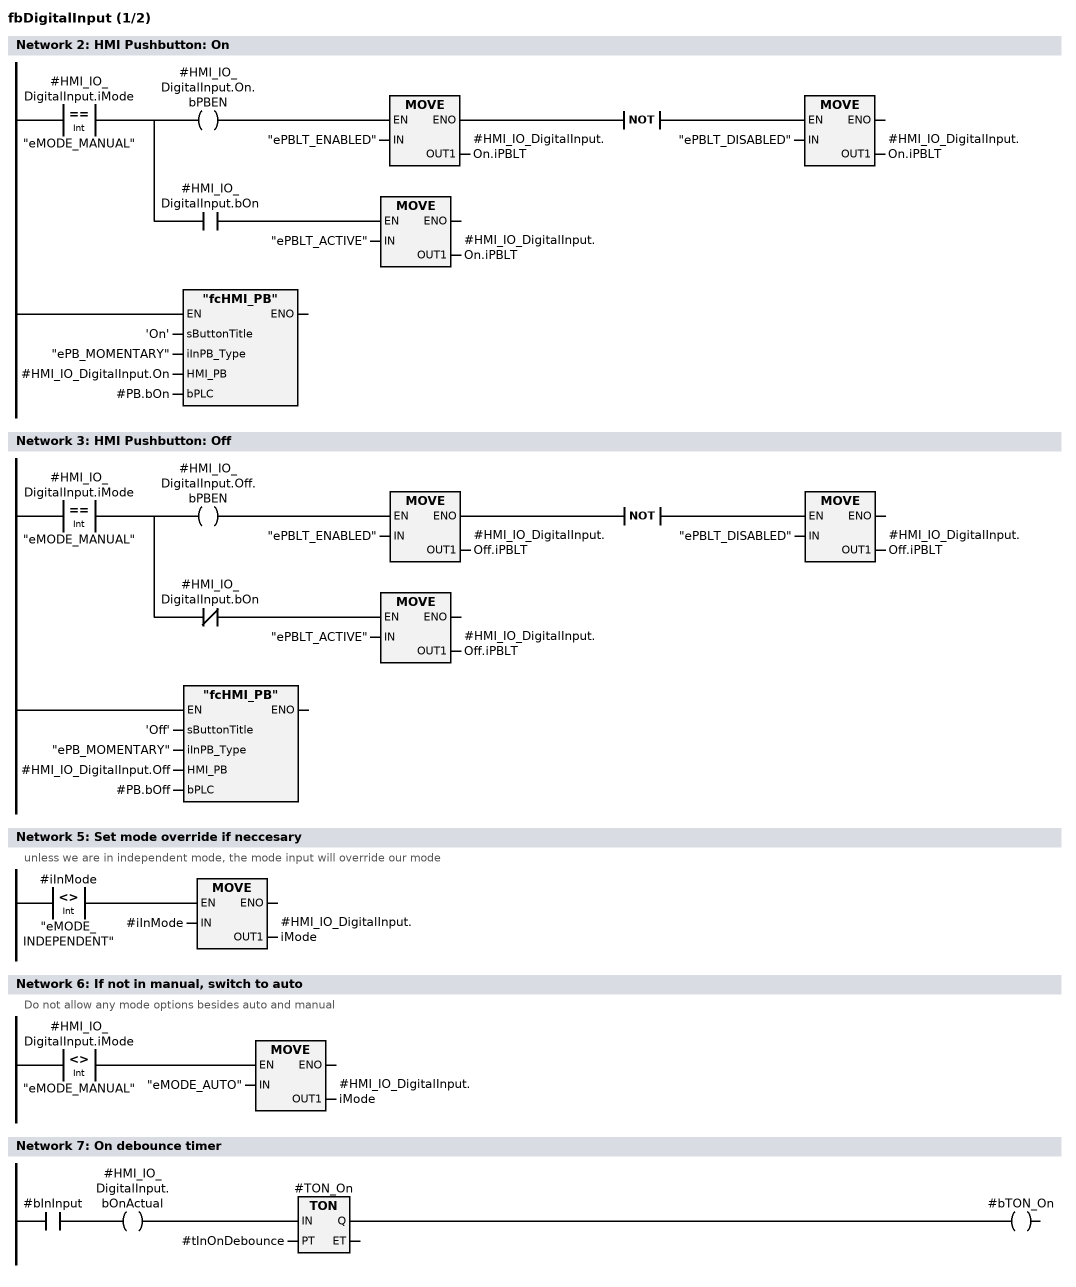
   RUNG wire#powerrail
      { S7_Templates := "SrcType := Int" } EQ_Contact(in1 := #HMI_IO_DigitalInput.iMode, in2 := "eMODE_MANUAL")
      wire#w1
      Coil( #HMI_IO_DigitalInput.On.bPBEN )
      Move(in := "ePBLT_ENABLED", out1 => #HMI_IO_DigitalInput.On.iPBLT)
      Not()
      Move(in := "ePBLT_DISABLED", out1 => #HMI_IO_DigitalInput.On.iPBLT)
   END_RUNG
   RUNG wire#w1
      Contact( #HMI_IO_DigitalInput.bOn )
      Move(in := "ePBLT_ACTIVE", out1 => #HMI_IO_DigitalInput.On.iPBLT)
   END_RUNG
   RUNG wire#powerrail
      "fcHMI_PB"(sButtonTitle := 'On', iInPB_Type := "ePB_MOMENTARY", HMI_PB := #HMI_IO_DigitalInput.On, bPLC := #PB.bOn)
   END_RUNG
   // the same network as SCL:
   #HMI_IO_DigitalInput.On.bPBEN := #HMI_IO_DigitalInput.iMode = "eMODE_MANUAL";
   IF #HMI_IO_DigitalInput.On.bPBEN THEN #HMI_IO_DigitalInput.On.iPBLT := "ePBLT_ENABLED"; END_IF;
   IF NOT #HMI_IO_DigitalInput.On.bPBEN THEN #HMI_IO_DigitalInput.On.iPBLT := "ePBLT_DISABLED"; END_IF;
   IF #HMI_IO_DigitalInput.On.bPBEN AND #HMI_IO_DigitalInput.bOn THEN
       #HMI_IO_DigitalInput.On.iPBLT := "ePBLT_ACTIVE";
   END_IF;
   "fcHMI_PB"(sButtonTitle := 'On',
              iInPB_Type := "ePB_MOMENTARY",
              HMI_PB := #HMI_IO_DigitalInput.On,
              bPLC := #PB.bOn);
END_REGION

REGION Network 3: HMI Pushbutton: Off
   RUNG wire#powerrail
      { S7_Templates := "SrcType := Int" } EQ_Contact(in1 := #HMI_IO_DigitalInput.iMode, in2 := "eMODE_MANUAL")
      wire#w1
      Coil( #HMI_IO_DigitalInput.Off.bPBEN )
      Move(in := "ePBLT_ENABLED", out1 => #HMI_IO_DigitalInput.Off.iPBLT)
      Not()
      Move(in := "ePBLT_DISABLED", out1 => #HMI_IO_DigitalInput.Off.iPBLT)
   END_RUNG
   RUNG wire#w1
      I_Contact( #HMI_IO_DigitalInput.bOn )
      Move(in := "ePBLT_ACTIVE", out1 => #HMI_IO_DigitalInput.Off.iPBLT)
   END_RUNG
   RUNG wire#powerrail
      "fcHMI_PB"(sButtonTitle := 'Off', iInPB_Type := "ePB_MOMENTARY", HMI_PB := #HMI_IO_DigitalInput.Off, bPLC := #PB.bOff)
   END_RUNG
   // the same network as SCL:
   #HMI_IO_DigitalInput.Off.bPBEN := #HMI_IO_DigitalInput.iMode = "eMODE_MANUAL";
   IF #HMI_IO_DigitalInput.Off.bPBEN THEN #HMI_IO_DigitalInput.Off.iPBLT := "ePBLT_ENABLED"; END_IF;
   IF NOT #HMI_IO_DigitalInput.Off.bPBEN THEN #HMI_IO_DigitalInput.Off.iPBLT := "ePBLT_DISABLED"; END_IF;
   IF #HMI_IO_DigitalInput.Off.bPBEN AND NOT #HMI_IO_DigitalInput.bOn THEN
       #HMI_IO_DigitalInput.Off.iPBLT := "ePBLT_ACTIVE";
   END_IF;
   "fcHMI_PB"(sButtonTitle := 'Off',
              iInPB_Type := "ePB_MOMENTARY",
              HMI_PB := #HMI_IO_DigitalInput.Off,
              bPLC := #PB.bOff);
END_REGION

REGION Network 4: --------------------------------------------------- Control Logic ------------------------------------------------------------
END_REGION

REGION Network 5: Set mode override if neccesary
   // unless we are in independent mode, the mode input will override our mode
   RUNG wire#powerrail
      { S7_Templates := "SrcType := Int" } NE_Contact(in1 := #iInMode, in2 := "eMODE_INDEPENDENT")
      { S7_GenerateENO := "TRUE" } Move(in := #iInMode, out1 => #HMI_IO_DigitalInput.iMode)
   END_RUNG
   // the same network as SCL:
   IF #iInMode <> "eMODE_INDEPENDENT" THEN #HMI_IO_DigitalInput.iMode := #iInMode; END_IF;
END_REGION

REGION Network 6: If not in manual, switch to auto
   // Do not allow any mode options besides auto and manual
   RUNG wire#powerrail
      { S7_Templates := "SrcType := Int" } NE_Contact(in1 := #HMI_IO_DigitalInput.iMode, in2 := "eMODE_MANUAL")
      Move(in := "eMODE_AUTO", out1 => #HMI_IO_DigitalInput.iMode)
   END_RUNG
   // the same network as SCL:
   IF #HMI_IO_DigitalInput.iMode <> "eMODE_MANUAL" THEN #HMI_IO_DigitalInput.iMode := "eMODE_AUTO"; END_IF;
END_REGION

REGION Network 7: On debounce timer
   #HMI_IO_DigitalInput.bOnActual := #bInInput;
   #TON_On.TON(IN := #bInInput, PT := #tInOnDebounce);
   #bTON_On := #TON_On.Q;
END_REGION

REGION Network 8: On logic
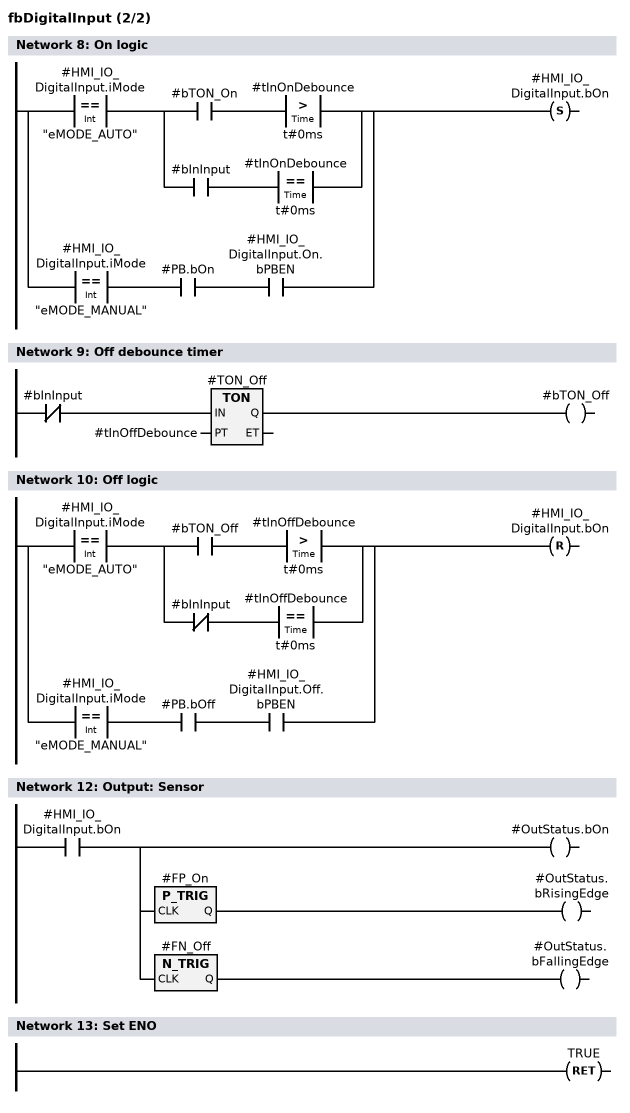
   RUNG wire#powerrail
      { S7_Templates := "SrcType := Int" } EQ_Contact(in1 := #HMI_IO_DigitalInput.iMode, in2 := "eMODE_AUTO")
      wire#w1
      Contact( #bTON_On )
      { S7_Templates := "SrcType := Time" } GT_Contact(in1 := #tInOnDebounce, in2 := t#0ms)
      wire#w2
      S_Coil( #HMI_IO_DigitalInput.bOn )
   END_RUNG
   RUNG wire#w1
      Contact( #bInInput )
      { S7_Templates := "SrcType := Time" } EQ_Contact(in1 := #tInOnDebounce, in2 := t#0ms)
   END_RUNG wire#w2
   RUNG wire#powerrail
      { S7_Templates := "SrcType := Int" } EQ_Contact(in1 := #HMI_IO_DigitalInput.iMode, in2 := "eMODE_MANUAL")
      Contact( #PB.bOn )
      Contact( #HMI_IO_DigitalInput.On.bPBEN )
   END_RUNG wire#w2
   // the same network as SCL:
   IF ((#HMI_IO_DigitalInput.iMode = "eMODE_AUTO") AND ((#bTON_On AND (#tInOnDebounce > t#0ms)) OR (#bInInput AND (#tInOnDebounce = t#0ms)))) OR ((#HMI_IO_DigitalInput.iMode = "eMODE_MANUAL") AND #PB.bOn AND #HMI_IO_DigitalInput.On.bPBEN) THEN
       #HMI_IO_DigitalInput.bOn := TRUE;
   END_IF;
END_REGION

REGION Network 9: Off debounce timer
   #TON_Off.TON(IN := NOT #bInInput, PT := #tInOffDebounce);
   #bTON_Off := #TON_Off.Q;
END_REGION

REGION Network 10: Off logic
   RUNG wire#powerrail
      { S7_Templates := "SrcType := Int" } EQ_Contact(in1 := #HMI_IO_DigitalInput.iMode, in2 := "eMODE_AUTO")
      wire#w1
      Contact( #bTON_Off )
      { S7_Templates := "SrcType := Time" } GT_Contact(in1 := #tInOffDebounce, in2 := t#0ms)
      wire#w2
      R_Coil( #HMI_IO_DigitalInput.bOn )
   END_RUNG
   RUNG wire#w1
      I_Contact( #bInInput )
      { S7_Templates := "SrcType := Time" } EQ_Contact(in1 := #tInOffDebounce, in2 := t#0ms)
   END_RUNG wire#w2
   RUNG wire#powerrail
      { S7_Templates := "SrcType := Int" } EQ_Contact(in1 := #HMI_IO_DigitalInput.iMode, in2 := "eMODE_MANUAL")
      Contact( #PB.bOff )
      Contact( #HMI_IO_DigitalInput.Off.bPBEN )
   END_RUNG wire#w2
   // the same network as SCL:
   IF ((#HMI_IO_DigitalInput.iMode = "eMODE_AUTO") AND ((#bTON_Off AND (#tInOffDebounce > t#0ms)) OR (NOT #bInInput AND (#tInOffDebounce = t#0ms)))) OR ((#HMI_IO_DigitalInput.iMode = "eMODE_MANUAL") AND #PB.bOff AND #HMI_IO_DigitalInput.Off.bPBEN) THEN
       #HMI_IO_DigitalInput.bOn := FALSE;
   END_IF;
END_REGION

REGION Network 11: --------------------------------------------------------- Outputs ------------------------------------------------------------------
END_REGION

REGION Network 12: Output: Sensor
   RUNG wire#powerrail
      Contact( #HMI_IO_DigitalInput.bOn )
      wire#w1
      Coil( #OutStatus.bOn )
   END_RUNG
   RUNG wire#w1
      P_Trig( #FP_On )
      Coil( #OutStatus.bRisingEdge )
   END_RUNG
   RUNG wire#w1
      N_Trig( #FN_Off )
      Coil( #OutStatus.bFallingEdge )
   END_RUNG
   // the same network as SCL:
   #OutStatus.bOn := #HMI_IO_DigitalInput.bOn;
   #_w1 := #HMI_IO_DigitalInput.bOn AND NOT #FP_On;   // rising edge
   #FP_On := #HMI_IO_DigitalInput.bOn;
   #OutStatus.bRisingEdge := #_w1;
   #_w2 := NOT #HMI_IO_DigitalInput.bOn AND #FN_Off;   // falling edge
   #FN_Off := #HMI_IO_DigitalInput.bOn;
   #OutStatus.bFallingEdge := #_w2;
END_REGION

REGION Network 13: Set ENO
   RUNG wire#powerrail
      ReturnCoil( TRUE )
   END_RUNG
   // the same network as SCL:
   ENO := TRUE;
   RETURN;
END_REGION
END_FUNCTION_BLOCK

// folder: 5 - LIBRARY/Resources/HMI

FUNCTION "fcHMI_PB" : Void   // FC1030, LAD
TITLE = fcHMI_PB
{ S7_Optimized_Access := 'FALSE' }
VERSION : 0.1
// Used for HMI push buttons that handshake between the HMI and PLC (PB HMI bits are set by the HMI, and reset by the PLC).
   VAR_INPUT
      sButtonTitle : String;
      iInPB_Type : Int;   // Momentary, Maintained, or Latch
   END_VAR
   VAR_IN_OUT
      HMI_PB : "udtHMI_PushButton";
      bPLC : Bool;
   END_VAR
   VAR_TEMP   // added for the SCL form of the ladder/FBD networks
      _w1 : Bool;
      _w2 : Bool;
      _w3 : Bool;
      _w4 : Bool;
   END_VAR
BEGIN

REGION Network 1: Transfer button title for display on the HMI
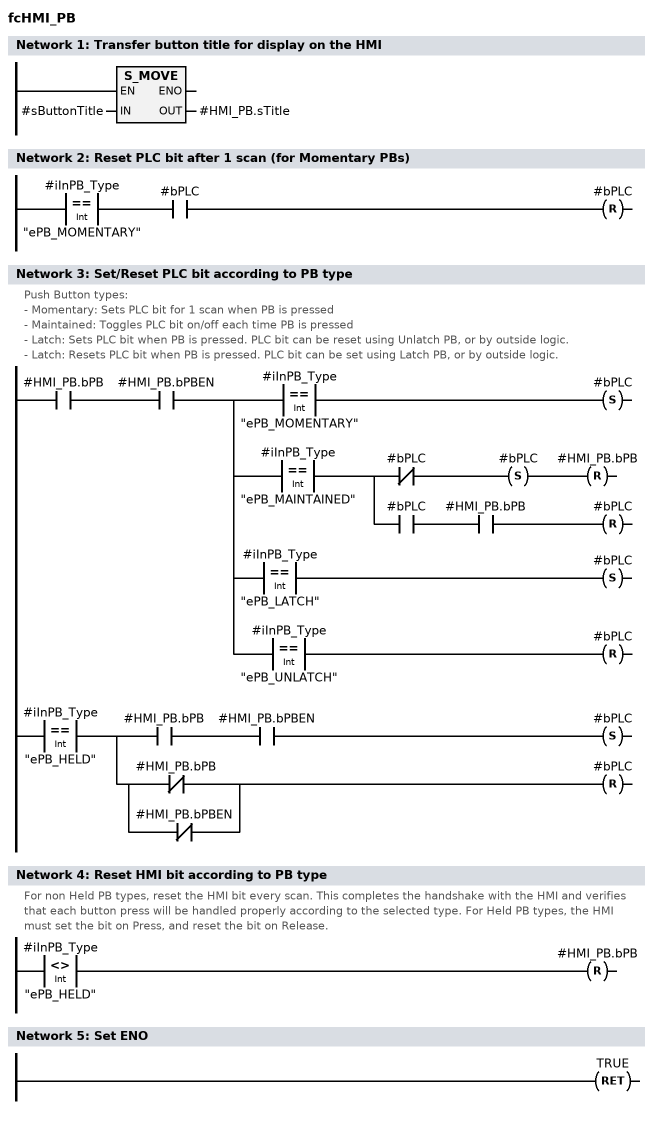
   RUNG wire#powerrail
      S_Move(in := #sButtonTitle, out => #HMI_PB.sTitle)
   END_RUNG
   // the same network as SCL:
   #HMI_PB.sTitle := #sButtonTitle;
END_REGION

REGION Network 2: Reset PLC bit after 1 scan (for Momentary PBs)
   RUNG wire#powerrail
      { S7_Templates := "SrcType := Int" } EQ_Contact(in1 := #iInPB_Type, in2 := "ePB_MOMENTARY")
      Contact( #bPLC )
      R_Coil( #bPLC )
   END_RUNG
   // the same network as SCL:
   IF (#iInPB_Type = "ePB_MOMENTARY") AND #bPLC THEN #bPLC := FALSE; END_IF;
END_REGION

REGION Network 3: Set/Reset PLC bit according to PB type
   // Push Button types:
   // - Momentary: Sets PLC bit for 1 scan when PB is pressed
   // - Maintained: Toggles PLC bit on/off each time PB is pressed
   // - Latch: Sets PLC bit when PB is pressed. PLC bit can be reset using Unlatch PB, or by outside logic.
   // - Latch: Resets PLC bit when PB is pressed. PLC bit can be set using Latch PB, or by outside logic.
   RUNG wire#powerrail
      Contact( #HMI_PB.bPB )
      Contact( #HMI_PB.bPBEN )
      wire#w1
      { S7_Templates := "SrcType := Int" } EQ_Contact(in1 := #iInPB_Type, in2 := "ePB_MOMENTARY")
      S_Coil( #bPLC )
   END_RUNG
   RUNG wire#w1
      { S7_Templates := "SrcType := Int" } EQ_Contact(in1 := #iInPB_Type, in2 := "ePB_MAINTAINED")
      wire#w2
      I_Contact( #bPLC )
      S_Coil( #bPLC )
      R_Coil( #HMI_PB.bPB )
   END_RUNG
   RUNG wire#w2
      Contact( #bPLC )
      Contact( #HMI_PB.bPB )
      R_Coil( #bPLC )
   END_RUNG
   RUNG wire#w1
      { S7_Templates := "SrcType := Int" } EQ_Contact(in1 := #iInPB_Type, in2 := "ePB_LATCH")
      S_Coil( #bPLC )
   END_RUNG
   RUNG wire#w1
      { S7_Templates := "SrcType := Int" } EQ_Contact(in1 := #iInPB_Type, in2 := "ePB_UNLATCH")
      R_Coil( #bPLC )
   END_RUNG
   RUNG wire#powerrail
      { S7_Templates := "SrcType := Int" } EQ_Contact(in1 := #iInPB_Type, in2 := "ePB_HELD")
      wire#w3
      Contact( #HMI_PB.bPB )
      Contact( #HMI_PB.bPBEN )
      S_Coil( #bPLC )
   END_RUNG
   RUNG wire#w3
      I_Contact( #HMI_PB.bPB )
      wire#w4
      R_Coil( #bPLC )
   END_RUNG
   RUNG wire#w3
      I_Contact( #HMI_PB.bPBEN )
   END_RUNG wire#w4
   // the same network as SCL:
   #_w1 := #HMI_PB.bPB AND #HMI_PB.bPBEN;
   IF #_w1 AND (#iInPB_Type = "ePB_MOMENTARY") THEN #bPLC := TRUE; END_IF;
   #_w2 := #_w1 AND (#iInPB_Type = "ePB_MAINTAINED");
   #_w3 := #_w2 AND NOT #bPLC;
   IF #_w3 THEN
       #bPLC := TRUE;
       #HMI_PB.bPB := FALSE;
   END_IF;
   IF #_w2 AND #bPLC AND #HMI_PB.bPB THEN #bPLC := FALSE; END_IF;
   IF #_w1 AND (#iInPB_Type = "ePB_LATCH") THEN #bPLC := TRUE; END_IF;
   IF #_w1 AND (#iInPB_Type = "ePB_UNLATCH") THEN #bPLC := FALSE; END_IF;
   #_w4 := #iInPB_Type = "ePB_HELD";
   IF #_w4 AND #HMI_PB.bPB AND #HMI_PB.bPBEN THEN #bPLC := TRUE; END_IF;
   IF #_w4 AND (NOT #HMI_PB.bPB OR NOT #HMI_PB.bPBEN) THEN #bPLC := FALSE; END_IF;
END_REGION

REGION Network 4: Reset HMI bit according to PB type
   // For non Held PB types, reset the HMI bit every scan. This completes the handshake with the HMI and verifies that each button press will be handled properly according to the selected type. For Held PB types, the HMI must set the bit on Press, and reset the bit on Release.
   RUNG wire#powerrail
      { S7_Templates := "SrcType := Int" } NE_Contact(in1 := #iInPB_Type, in2 := "ePB_HELD")
      R_Coil( #HMI_PB.bPB )
   END_RUNG
   // the same network as SCL:
   IF #iInPB_Type <> "ePB_HELD" THEN #HMI_PB.bPB := FALSE; END_IF;
END_REGION

REGION Network 5: Set ENO
   RUNG wire#powerrail
      ReturnCoil( TRUE )
   END_RUNG
   // the same network as SCL:
   ENO := TRUE;
   RETURN;
END_REGION
END_FUNCTION

// folder: Open Library V14 SP1/Resources/Conversion

FUNCTION "fcSwapBytes" : Void   // FC304, LAD
TITLE = Swap the bytes in a word
{ S7_Optimized_Access := 'TRUE' }
AUTHOR : DMC
FAMILY : LowLevel
VERSION : 0.1
// High byte and Low Byte are swapped
   VAR_INPUT
      wInWord : Word;   // Word to be swapped
   END_VAR
   VAR_OUTPUT
      wOutWord : Word;
   END_VAR
BEGIN

REGION Network 1: Swap the bytes
   // High byte and Low Byte are swapped
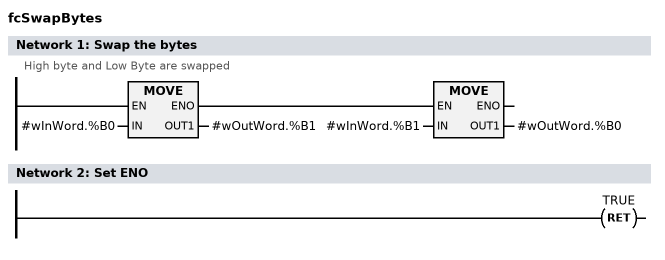
   RUNG wire#powerrail
      { S7_GenerateENO := "TRUE" } Move(in := #wInWord.%B0, out1 => #wOutWord.%B1)
      { S7_GenerateENO := "TRUE" } Move(in := #wInWord.%B1, out1 => #wOutWord.%B0)
   END_RUNG
   // the same network as SCL:
   // ENO of a box is taken as its EN; it also drops when the box reports an error
   #wOutWord.%B1 := #wInWord.%B0;
   #wOutWord.%B0 := #wInWord.%B1;
END_REGION

REGION Network 2: Set ENO
   RUNG wire#powerrail
      ReturnCoil( TRUE )
   END_RUNG
   // the same network as SCL:
   ENO := TRUE;
   RETURN;
END_REGION
END_FUNCTION

// folder: Open Library V14 SP1/Resources/IO

FUNCTION "fcReadInput" : Void   // FC350, LAD
TITLE = Read/Scale input word
{ S7_Optimized_Access := 'TRUE' }
AUTHOR : DMC
FAMILY : IO
VERSION : 0.1
   VAR_INPUT
      wInValue : Word;   // Input from I/O module
      iInRawMax : Int;   // Raw maximum - overflow limit
      iInRawMin : Int;   // Raw minimum - underflow limit
      rInScaledMax : Real;   // Engineering units range max
      rInScaledMin : Real;   // Engineering units range min
      bInSwapBytes : Bool;
      bInErrorReset : Bool;
   END_VAR
   VAR_OUTPUT
      rOutValue : Real;
   END_VAR
   VAR_IN_OUT
      bOutError : Bool;
   END_VAR
   VAR_TEMP
      wTemp : Word;
      wInputValue : Word;
      iInputValue : Int;
      diTemp : DInt;
      rTemp : Real;
      rPreScaledVal : Real;
      rPreScaledRange : Real;
      rScaledOut : Real;
      rRawMax : Real;
      rRawMin : Real;
      rScaledRange : Real;
   END_VAR
BEGIN

REGION Network 1: Swap input value bytes if needed
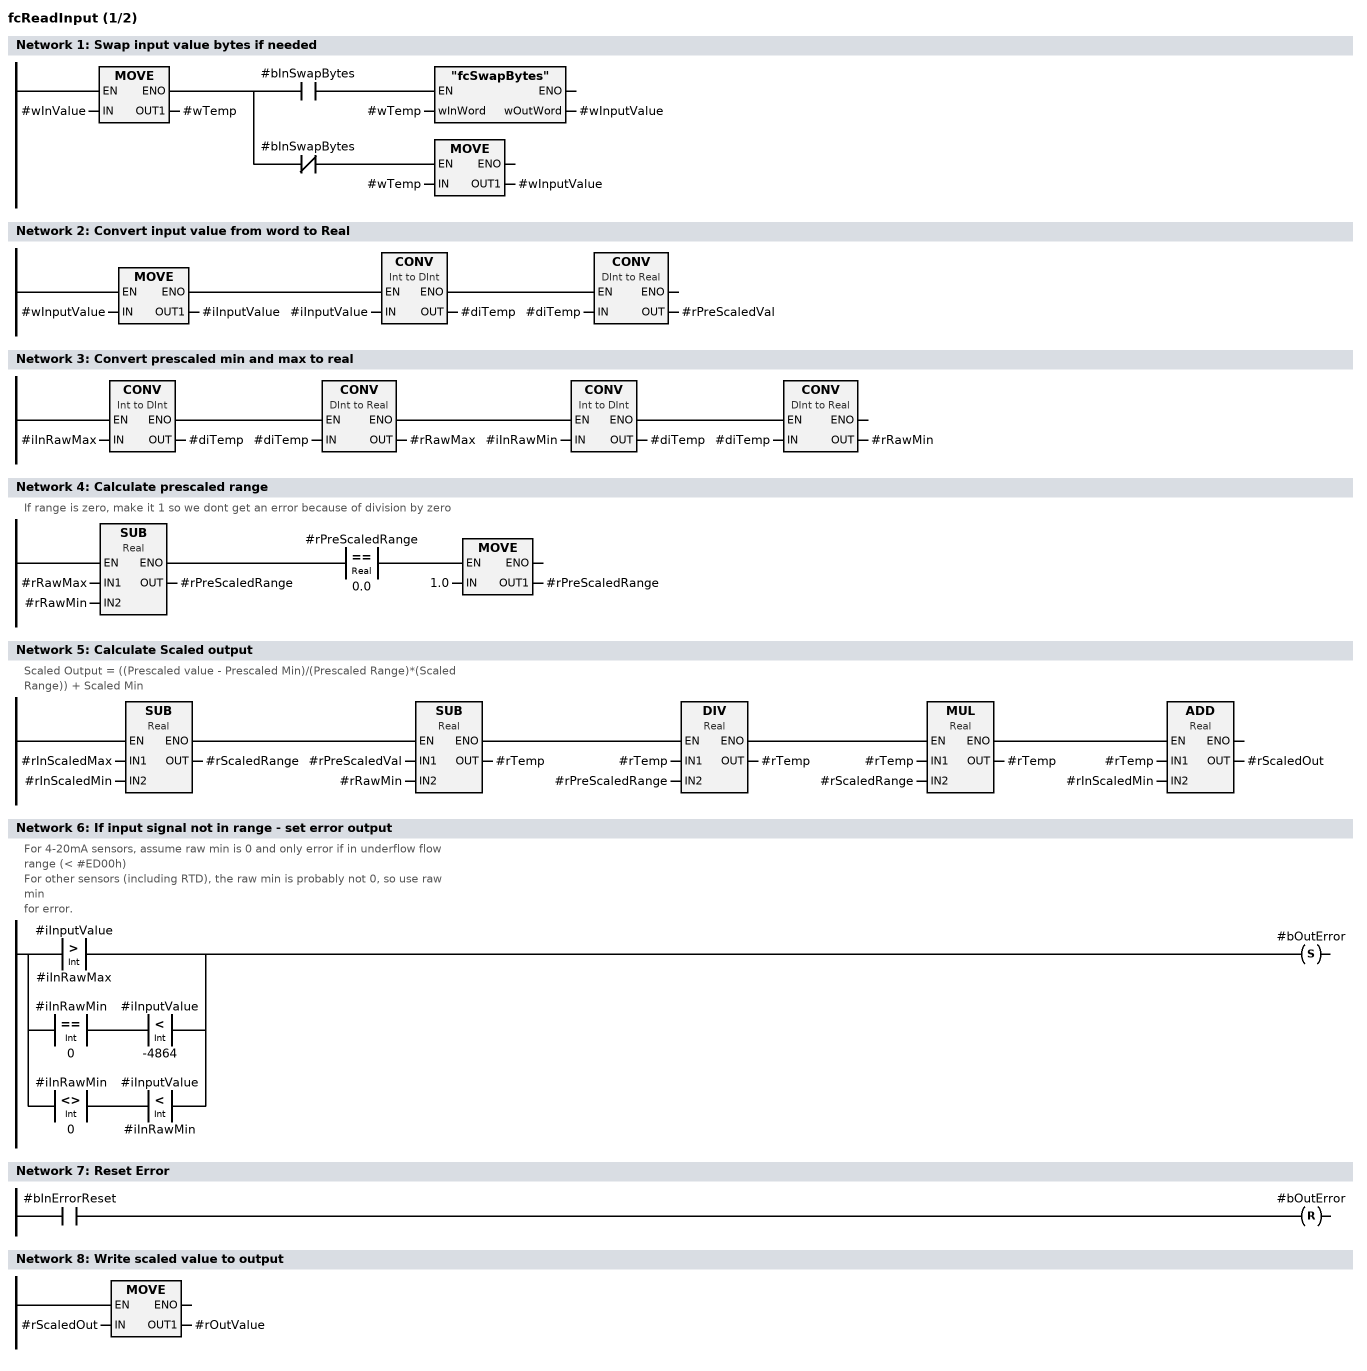
   RUNG wire#powerrail
      { S7_GenerateENO := "TRUE" } Move(in := #wInValue, out1 => #wTemp)
      wire#w1
      Contact( #bInSwapBytes )
      "fcSwapBytes"(wInWord := #wTemp, wOutWord => #wInputValue)
   END_RUNG
   RUNG wire#w1
      I_Contact( #bInSwapBytes )
      { S7_GenerateENO := "TRUE" } Move(in := #wTemp, out1 => #wInputValue)
   END_RUNG
   // the same network as SCL:
   // ENO of a box is taken as its EN; it also drops when the box reports an error
   #wTemp := #wInValue;
   IF #bInSwapBytes THEN "fcSwapBytes"(wInWord := #wTemp, wOutWord => #wInputValue); END_IF;
   IF NOT #bInSwapBytes THEN #wInputValue := #wTemp; END_IF;
END_REGION

REGION Network 2: Convert input value from word to Real
   RUNG wire#powerrail
      { S7_GenerateENO := "TRUE" } Move(in := #wInputValue, out1 => #iInputValue)
      { S7_Templates := "[SrcType := Int, DestType := DInt]"; S7_GenerateENO := "TRUE" } Convert(in := #iInputValue, out => #diTemp)
      { S7_Templates := "[SrcType := DInt, DestType := Real]"; S7_GenerateENO := "TRUE" } Convert(in := #diTemp, out => #rPreScaledVal)
   END_RUNG
   // the same network as SCL:
   // ENO of a box is taken as its EN; it also drops when the box reports an error
   #iInputValue := #wInputValue;
   #diTemp := INT_TO_DINT(#iInputValue);
   #rPreScaledVal := DINT_TO_REAL(#diTemp);
END_REGION

REGION Network 3: Convert prescaled min and max to real
   RUNG wire#powerrail
      { S7_Templates := "[SrcType := Int, DestType := DInt]"; S7_GenerateENO := "TRUE" } Convert(in := #iInRawMax, out => #diTemp)
      { S7_Templates := "[SrcType := DInt, DestType := Real]"; S7_GenerateENO := "TRUE" } Convert(in := #diTemp, out => #rRawMax)
      { S7_Templates := "[SrcType := Int, DestType := DInt]"; S7_GenerateENO := "TRUE" } Convert(in := #iInRawMin, out => #diTemp)
      { S7_Templates := "[SrcType := DInt, DestType := Real]"; S7_GenerateENO := "TRUE" } Convert(in := #diTemp, out => #rRawMin)
   END_RUNG
   // the same network as SCL:
   // ENO of a box is taken as its EN; it also drops when the box reports an error
   #diTemp := INT_TO_DINT(#iInRawMax);
   #rRawMax := DINT_TO_REAL(#diTemp);
   #diTemp := INT_TO_DINT(#iInRawMin);
   #rRawMin := DINT_TO_REAL(#diTemp);
END_REGION

REGION Network 4: Calculate prescaled range
   // If range is zero, make it 1 so we dont get an error because of division by zero
   RUNG wire#powerrail
      { S7_Templates := "SrcType := Real"; S7_GenerateENO := "TRUE" } Sub(in1 := #rRawMax, in2 := #rRawMin, out => #rPreScaledRange)
      { S7_Templates := "SrcType := Real" } EQ_Contact(in1 := #rPreScaledRange, in2 := 0.0)
      { S7_GenerateENO := "TRUE" } Move(in := 1.0, out1 => #rPreScaledRange)
   END_RUNG
   // the same network as SCL:
   // ENO of a box is taken as its EN; it also drops when the box reports an error
   #rPreScaledRange := #rRawMax - #rRawMin;
   IF #rPreScaledRange = 0.0 THEN #rPreScaledRange := 1.0; END_IF;
END_REGION

REGION Network 5: Calculate Scaled output
   // Scaled Output = ((Prescaled value - Prescaled Min)/(Prescaled Range)*(Scaled 
   // Range)) + Scaled Min
   RUNG wire#powerrail
      { S7_Templates := "SrcType := Real"; S7_GenerateENO := "TRUE" } Sub(in1 := #rInScaledMax, in2 := #rInScaledMin, out => #rScaledRange)
      { S7_Templates := "SrcType := Real"; S7_GenerateENO := "TRUE" } Sub(in1 := #rPreScaledVal, in2 := #rRawMin, out => #rTemp)
      { S7_Templates := "SrcType := Real"; S7_GenerateENO := "TRUE" } Div(in1 := #rTemp, in2 := #rPreScaledRange, out => #rTemp)
      { S7_Templates := "SrcType := Real"; S7_GenerateENO := "TRUE" } Mul(in1 := #rTemp, in2 := #rScaledRange, out => #rTemp)
      { S7_Templates := "SrcType := Real"; S7_GenerateENO := "TRUE" } Add(in1 := #rTemp, in2 := #rInScaledMin, out => #rScaledOut)
   END_RUNG
   // the same network as SCL:
   // ENO of a box is taken as its EN; it also drops when the box reports an error
   #rScaledRange := #rInScaledMax - #rInScaledMin;
   #rTemp := #rPreScaledVal - #rRawMin;
   #rTemp := #rTemp / #rPreScaledRange;
   #rTemp := #rTemp * #rScaledRange;
   #rScaledOut := #rTemp + #rInScaledMin;
END_REGION

REGION Network 6: If input signal not in range - set error output
   // For 4-20mA sensors, assume raw min is 0 and only error if in underflow flow 
   // range (< #ED00h)
   // 
   // For other sensors (including RTD), the raw min is probably not 0, so use raw 
   // min 
   // for error.
   RUNG wire#powerrail
      { S7_Templates := "SrcType := Int" } GT_Contact(in1 := #iInputValue, in2 := #iInRawMax)
      wire#w1
      S_Coil( #bOutError )
   END_RUNG
   RUNG wire#powerrail
      { S7_Templates := "SrcType := Int" } EQ_Contact(in1 := #iInRawMin, in2 := 0)
      { S7_Templates := "SrcType := Int" } LT_Contact(in1 := #iInputValue, in2 := -4864)
   END_RUNG wire#w1
   RUNG wire#powerrail
      { S7_Templates := "SrcType := Int" } NE_Contact(in1 := #iInRawMin, in2 := 0)
      { S7_Templates := "SrcType := Int" } LT_Contact(in1 := #iInputValue, in2 := #iInRawMin)
   END_RUNG wire#w1
   // the same network as SCL:
   IF (#iInputValue > #iInRawMax) OR ((#iInRawMin = 0) AND (#iInputValue < (-4864))) OR ((#iInRawMin <> 0) AND (#iInputValue < #iInRawMin)) THEN
       #bOutError := TRUE;
   END_IF;
END_REGION

REGION Network 7: Reset Error
   RUNG wire#powerrail
      Contact( #bInErrorReset )
      R_Coil( #bOutError )
   END_RUNG
   // the same network as SCL:
   IF #bInErrorReset THEN #bOutError := FALSE; END_IF;
END_REGION

REGION Network 8: Write scaled value to output
   RUNG wire#powerrail
      { S7_GenerateENO := "TRUE" } Move(in := #rScaledOut, out1 => #rOutValue)
   END_RUNG
   // the same network as SCL:
   #rOutValue := #rScaledOut;
END_REGION

REGION Network 9: Set ENO
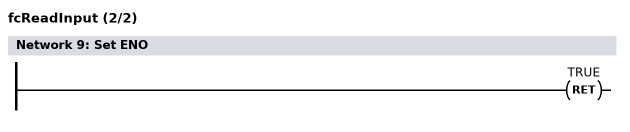
   RUNG wire#powerrail
      ReturnCoil( TRUE )
   END_RUNG
   // the same network as SCL:
   ENO := TRUE;
   RETURN;
END_REGION
END_FUNCTION

(* ===== HMI "HMI_RT_1" =====

ScreenModuleEditorView "DO_Faceplate" 640x480
   Circle "Circle_1" at 175,10 size 48x48
      Appearance <- "bStatus"
   Switch "Switch_1" at 10,10 size 95x48; TextOn 'ON'; CaptionText 'Switch'; TextOff 'OFF'
      ProcessValue <- "bCommand"
*)

(* ===== HMI "HMI_RT_1" =====

ScreenModuleEditorView "AI_Faceplate" 640x480
   TextField "Text field_1" at 10,13 size 17x25; Text 'Text'
   IOField "I/O field_1" at 236,10 size 96x32; FormatPattern 9999999
      ProcessValue <- "Property_1.rInputValue"
   IOField "I/O field_2" at 374,10 size 152x32; FormatPattern 99999.99
      ProcessValue <- "Property_1.rActiveValue"
*)

(* ===== HMI "HMI_RT_1" =====

ScreenModuleEditorView "AI_Faceplate" 640x480
   TextField "Text field_1" at 10,13 size 17x25; Text 'Text'
   IOField "I/O field_1" at 236,10 size 96x32; FormatPattern 9999999
      ProcessValue <- "Property_1.rInputValue"
   IOField "I/O field_2" at 374,10 size 152x32; FormatPattern 99999.99
      ProcessValue <- "Property_1.rActiveValue"
*)

(* ===== HMI "HMI_RT_1" =====

ScreenModuleEditorView "fpVFD_Motor_Horizontal" 640x480
   Rectangle "Rectangle_3" at 159,68 size 180x100
      Visibility <- "HMI_VFDControl.iMode"
   SymbolLibrary "Symbol library_3" at 167,75 size 165x85
      Appearance <- "HMI_VFDControl.iStatus"
   GraphicView "Graphic view_1" at 210,78 size 80x80; Picture "Interlock"
      Visibility <- "HMI_VFDControl.bInterlock"
   Button "Button_1" at 159,68 size 181x101; TextOff 'Text'
*)

(* ===== HMI "HMI_RT_1" =====
system functions are stored by id; their names below are inferred from use

text list "InterlockList": 1 'Interlock Active'; 0 'Interlock Inactive'

text list "ErrorMessages": 0..1 'Status OK'; 1 'Motor Fault'

ScreenModuleEditorView "fpVFD_Popup" 640x480
   Button "Button_3" at 25,173 size 148x27; TextOff 'Start Forward'
      on Release: SetBit("HMI_VFDControl.bCommandForward")
      Appearance <- "HMI_VFDControl.bCommandForward"
      ObjectEnable <- "HMI_VFDControl.bCommandReverse"
   Button "Button_4" at 25,284 size 148x26; TextOff 'RESET'
      on Release: ResetBit("HMI_VFDControl.bResetError")
      on Press: SetBit("HMI_VFDControl.bResetError")
   Button "Button_6" at 25,203 size 148x28; TextOff 'Stop'
      on Release: ResetBit("HMI_VFDControl.bCommandForward"); ResetBit("HMI_VFDControl.bCommandReverse")
   Button "Button_7" at 25,235 size 148x28; TextOff 'Start Reverse'
      on Release: SetBit("HMI_VFDControl.bCommandReverse")
      Appearance <- "HMI_VFDControl.bCommandReverse"
      ObjectEnable <- "HMI_VFDControl.bCommandForward"
   TextField "Text field_5" at 42,53 size 42x15; Text 'Setpoint:'
   IOField "I/O field_2" at 88,51 size 91x18; FormatPattern 999.9; Unit  %
      ProcessValue <- "HMI_VFDControl.rTargetSpeed"
   TextField "Text field_7" at 21,91 size 63x15; Text 'Actual Speed:'
   IOField "I/O field_3" at 88,90 size 91x17; FormatPattern 999.9; Unit  %
      ProcessValue <- "HMI_VFDControl.rActualSpeed"
   SymbolicIOField "Symbolic I/O field_3" at 21,122 size 159x24; TextOn '1'; TextOff '0'; TextList "ErrorMessages"
      ProcessValue <- "HMI_VFDControl.bActiveError"
      Appearance <- "HMI_VFDControl.bActiveError"
   TextField "Text field_1" at 10,12 size 180x31; Text 'Motor ## VFD Control'
*)